TYPE LG_InputRegs :
STRUCT
	UI_ErrorCode		:	UINT;
	ui_OperationalMode	:	UINT;
	r_CoolantInletTemp	:	REAL;
	r_CoolantOutletTemp	:	REAL;
	r_BackupHeaterTemp	:	REAL;
	r_SWWTankTemp		:	REAL;
	r_SolarCollectorTemp:	REAL;
	r_RoomTemp1			:	REAL;
	r_FlowRate			:	REAL;
	r_FlowTempCircuit2	:	REAL;
	r_RoomTemp2			:	REAL;
	UI_EnergyStatus		:	UINT;
	r_OutsideTemp		:	REAL;		
END_STRUCT
END_TYPE

(* stored: Version 1.1.0.1, ProductVersion 3.1.4024.12
   DUT LG_InputRegs: Id {a7c214cc-f0ff-4a8b-8733-1fec05994e8b} *)
